// TwinCAT 3 PLC project Libraries2
// ProgramVersion: 3.1.4024.0
// libraries:
//   Tc2_Standard, * (Beckhoff Automation GmbH)
//   Tc2_System, * (Beckhoff Automation GmbH)
//   Tc3_Module, * (Beckhoff Automation GmbH)
//   Identical Library ,0.1.0.0,EuroSort
// project tree:
//   / PlcTask.TcTTO
//   POUs/ FB_TestFunctionBlock.TcPOU, MAIN.TcPOU
// real-time tasks:
//   TASK PlcTask: cycle T#10ms, priority 20, ADS port 350

CONFIGURATION Libraries2
    RESOURCE PLC ON TwinCAT3
        TASK PlcTask(INTERVAL := T#10ms, PRIORITY := 20);
        PROGRAM MAIN WITH PlcTask : MAIN;
    END_RESOURCE
END_CONFIGURATION

// ---- POUs/MAIN.TcPOU
PROGRAM MAIN
VAR
	fbO5D100 : Identical_Library.FB_O5D100;
	fbO5D100_2 : Identical_Library.FB_O5D100;
END_VAR

fbO5D100();
fbO5D100_2();

END_PROGRAM

// ---- POUs/FB_TestFunctionBlock.TcPOU
FUNCTION_BLOCK FB_TestFunctionBlock
VAR
	nCounter : LINT;
END_VAR

nCounter := nCounter + 1;

END_FUNCTION_BLOCK
